// SIMATIC S7-200 SMART project (STEP 7-Micro/WIN SMART), CPU SR20

SYMBOL_TABLE System Symbols
Clock_1s         SM0.5    // Clock pulse that is ON for 0.5 s, OFF for 0.5 s, for a duty cycle time of 1 s.
END_SYMBOL_TABLE

ORGANIZATION_BLOCK MAIN:OB1
TITLE=Program Comments
BEGIN
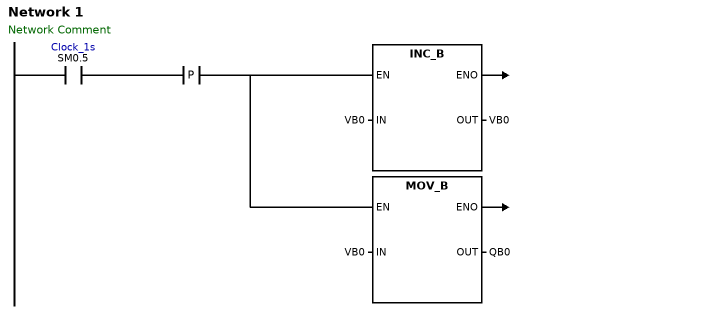
Network 1
// Network Comment
LD     Clock_1s:SM0.5
EU
INCB   VB0
MOVB   VB0, QB0
END_ORGANIZATION_BLOCK
